FUNCTION_BLOCK NORMAL_BEHAVIOUR_SIM
  {SET_ATTRIBUTE(OpcUa, SERVICE)}
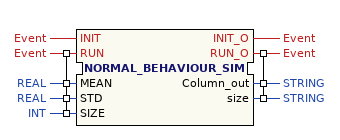
  EVENT_INPUT
    INIT;
    RUN WITH MEAN, STD, SIZE; {SET_ATTRIBUTE(OpcUa, Method)}
  END_EVENT
  EVENT_OUTPUT
    INIT_O;
    RUN_O WITH Column_out, size;
  END_EVENT
  VAR_INPUT
    MEAN : REAL; {SET_ATTRIBUTE(OpcUa, Variable.RUN)}
    STD : REAL; {SET_ATTRIBUTE(OpcUa, Variable.RUN)}
    SIZE : INT; {SET_ATTRIBUTE(OpcUa, Variable.RUN)}
  END_VAR
  VAR_OUTPUT
    Column_out : STRING; {SET_ATTRIBUTE(OpcUa, Variable.RUN)}
    size : STRING; {SET_ATTRIBUTE(OpcUa, Variable.RUN)}
  END_VAR
END_FUNCTION_BLOCK
